FUNCTION_BLOCK FB_PointingModelInversion
VAR_INPUT
	fAzimuth		: LREAL;	// current azimuth of telescope in degrees
	fElevation		: LREAL;		// current elevation of telescope in degrees
END_VAR
VAR_OUTPUT
	fAzimuthOffset		: LREAL;	// calculated azimuth offset of telescope in degrees
	fElevationOffset	: LREAL;	// calculated elevation offset of telescope in degrees
END_VAR
VAR
	i				: UINT;
	d_el			: LREAL := 0.0;
	d_az			: LREAL := 0.0;
	fElevationClamped	: LREAL;
	fbPointing		: REFERENCE TO FB_PointingModelForward;
END_VAR

d_el := 0.0;
d_az := 0.0;

// fbPointing is only ever set via FB_init(fbPointing := ...); nothing enforces that a consumer
// actually does, and calling through an unassigned REFERENCE TO crashes the whole PLC task (#7).
// Leave the offsets at 0.0 (no correction) rather than crash.
IF NOT __ISVALIDREF(fbPointing) THEN
	fAzimuthOffset := 0.0;
	fElevationOffset := 0.0;
	RETURN;
END_IF

// FB_PointingModelForward's own BNP/cos(el) term grows without bound approaching the zenith (89.9 deg is
// where the forward model switches to its own fixed clamp); feeding the iteration an elevation past that
// point keeps growing the offset further instead of converging to the bounded value the forward model
// would give at 89.9 deg
fElevationClamped := MIN(fElevation, 89.9);

// 2 passes converge to < 0.1" for every elevation/coefficient combination tried; 5 keeps a wide margin
// (needed for BROTLibTests' Inversion_Round_Trip, which checks self-consistency to 1e-9 deg)
FOR i:=0 TO 4 BY 1 DO
	fbPointing(
		fAzimuth   		 := fAzimuth   		  - d_az,
		fElevation 		 := fElevationClamped - d_el,
		fAzimuthOffset   => d_az,
		fElevationOffset => d_el,
	);
END_FOR;

fAzimuthOffset   := d_az;
fElevationOffset := d_el;

METHOD FB_init : BOOL
VAR_INPUT
	bInitRetains : BOOL; // if TRUE, the retain variables are initialized (warm start / cold start)
	bInCopyCode : BOOL;  // if TRUE, the instance afterwards gets moved into the copy code (online change)
	
	fbPointing		: REFERENCE TO FB_PointingModelForward;
END_VAR
THIS^.fbPointing REF= fbPointing;
END_METHOD

END_FUNCTION_BLOCK

(* stored: Version 1.1.0.1, ProductVersion 3.1.4024.15
   POU FB_PointingModelInversion: Id {414de569-9f94-41e7-a3f1-33de06319a3f}, SpecialFunc None
   Method FB_init: Id {c14393e7-a186-4c1a-a2ea-01e9bbbb0b43} *)
